KUKA KRL program: POUNCE.src, POUNCE.dat

--- POUNCE.src ---
&ACCESS RVP
&REL 1
&PARAM EDITMASK = *
DEF POUNCE( )
;FOLD INI
  ;FOLD BASISTECH INI
    GLOBAL INTERRUPT DECL 3 WHEN $STOPMESS==TRUE DO IR_STOPM ( )
    INTERRUPT ON 3
    BAS (#INITMOV,0 )
  ;ENDFOLD (BASISTECH INI)
  ;FOLD USER INI
    ;Make your modifications here

  ;ENDFOLD (USER INI)
;ENDFOLD (INI)
;********************************
; Gestamp Standards
; Line - Volvo
; Robot XXXXX
; Application - POUNCE
;********************************
; POUNCE
;********************************
;FOLD PTP P1 Vel=100 % PDAT1 Tool[1]:EOAT 1 Base[0];%{PE}%R 4.1.5,%MKUKATPBASIS,%CMOVE,%VPTP,%P 1:PTP, 2:P1, 3:, 5:100, 7:PDAT1
$BWDSTART=FALSE
PDAT_ACT=PPDAT1
BAS(#PTP_DAT)
FDAT_ACT=FP1
BAS(#FRAMES)
BAS(#VEL_PTP,100)
PTP XP1
;ENDFOLD
END

--- POUNCE.dat ---
&ACCESS RVP
&REL 1
&PARAM EDITMASK = *
DEFDAT POUNCE
;FOLD EXTERNAL DECLARATIONS;%{PE}%MKUKATPBASIS,%CEXT,%VCOMMON,%P
;FOLD BASISTECH EXT;%{PE}%MKUKATPBASIS,%CEXT,%VEXT,%P
EXT  BAS (BAS_COMMAND  :IN,REAL  :IN )
DECL INT SUCCESS
;ENDFOLD (BASISTECH EXT)
;FOLD USER EXT;%{E}%MKUKATPUSER,%CEXT,%VEXT,%P
;Make here your modifications

;ENDFOLD (USER EXT)
;ENDFOLD (EXTERNAL DECLARATIONS)
DECL E6AXIS XP1={A1 -0.224,A2 -136.109,A3 91.35,A4 0.0,A5 67.322,A6 -0.224,E1 0.0,E2 0.0,E3 0.0,E4 0.0,E5 0.0,E6 0.0}
DECL FDAT FP1={TOOL_NO 1,BASE_NO 0,IPO_FRAME #BASE}
DECL PDAT PPDAT1={VEL 100.0,ACC 100.0,APO_DIST 0.0}
ENDDAT
